(* CODESYS project Components.gvl.xml

Project tree, tasks and I/O mapping:
  global variables Components
*)

// Components
{attribute 'qualified_only'}
VAR_GLOBAL
	Agitator: Agitator;
	BagFeeder: BagFeeder;
	Door: Door;
	Heater: Heater;
	HeatSeal: HeatSeal;
	Hopper: Hopper;
	IceMaker: IceMaker;
	Kicker: Kicker;
END_VAR
